// TIA Portal V19 export
TYPE "C402_STU_IF_VKL_TYPIC"
   STRUCT
      COMM_OK { ExternalAccessible := 'False'; ExternalVisible := 'False'; ExternalWritable := 'False'} : Bool;   // Communicatie met 3B in werking
      CMD_ROOD { ExternalAccessible := 'False'; ExternalVisible := 'False'; ExternalWritable := 'False'} : Bool;   // Aansturing verkeerslicht Rood
      CMD_GROE { ExternalAccessible := 'False'; ExternalVisible := 'False'; ExternalWritable := 'False'} : Bool;   // Aansturing verkeerslicht Groen
      CMD_KNIP { ExternalAccessible := 'False'; ExternalVisible := 'False'; ExternalWritable := 'False'} : Bool;   // Aansturing verkeerslicht Geel Knipperen
      CMD_RES { ExternalAccessible := 'False'; ExternalVisible := 'False'; ExternalWritable := 'False'} : Bool;   // Reset van de latched storingen
      CMD_ONHD { ExternalAccessible := 'False'; ExternalVisible := 'False'; ExternalWritable := 'False'} : Bool;   // Automatische onderhoudstesten uitvoeren
      VGV_SNEL { ExternalAccessible := 'False'; ExternalVisible := 'False'; ExternalWritable := 'False'} : Bool;   // Vrijgave om versneld naar rood te gaan
   END_STRUCT;
END_TYPE
